(* Logix 5000 project; controller Modbus_TCP_Client_Example vendor 1 type 14 code 154 rev 32.15; software revision 32.05; part 10 of 10 *)
(* tags used below, declared in another part *)
   Transaction : raC_UDT_ModbusClientTransaction;
   Wrk_Bit : DINT;
   Wrk_Byte : DINT;
(* raC_Tec_NetModbusTCPClient_BuildReqStr, continued *)

ROUTINE Prescan   (* ladder *)
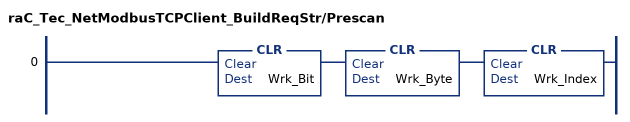
   0: CLR(Wrk_Bit)CLR(Wrk_Byte)CLR(Wrk_Index);
END_ROUTINE
END_ADD_ON_INSTRUCTION

ADD_ON_INSTRUCTION raC_Tec_NetModbusTCPClient_ChkWrReply   (* revision 2.0, ExecutePrescan *)
VAR_OUTPUT
   TransFound : BOOL; {access Read Only}
END_VAR
VAR_IN_OUT
   Transactions : raC_UDT_ModbusClientTransaction[5]; {required}
END_VAR
VAR_INPUT
   TransactionID : INT; {required}
   ModbusBytes : DINT; {required}
END_VAR
VAR_OUTPUT
   LocalOffset : INT; {access Read Only}
   Count : INT; {access Read Only}
END_VAR
VAR_INPUT
   Command : DINT; {required}
   LastTransaction : DINT; {required}
END_VAR
VAR
   Wrk_TransactionPtr : DINT; {access None}
END_VAR

ROUTINE Logic   (* ladder *)
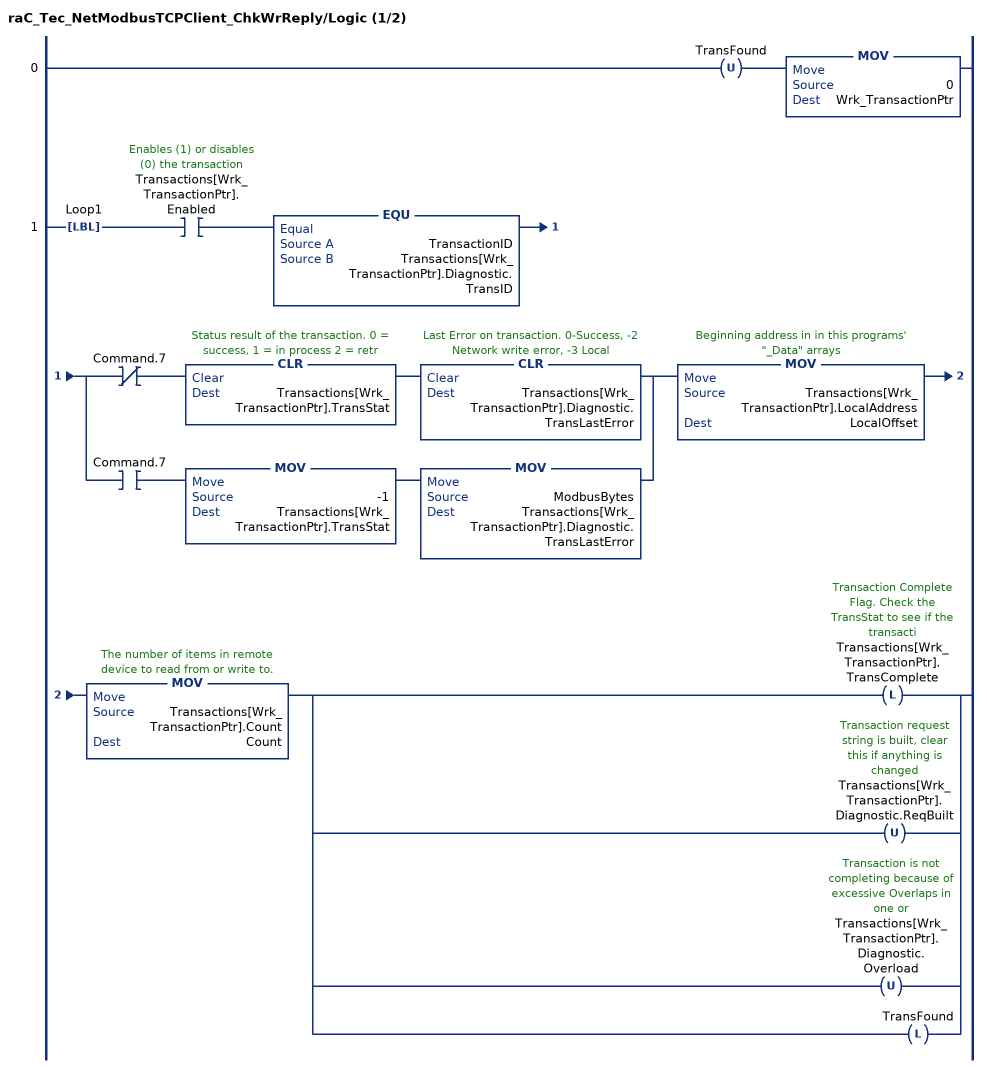
   0: OTU(TransFound)MOV(0,Wrk_TransactionPtr);
   1: LBL(Loop1)XIC(Transactions[Wrk_TransactionPtr].Enabled)EQU(TransactionID,Transactions[Wrk_TransactionPtr].Diagnostic.TransID)[XIO(Command.7) CLR(Transactions[Wrk_TransactionPtr].TransStat) CLR(Transactions[Wrk_TransactionPtr].Diagnostic.TransLastError) ,XIC(Command.7) MOV(-1,Transactions[Wrk_TransactionPtr].TransStat) MOV(ModbusBytes,Transactions[Wrk_TransactionPtr].Diagnostic.TransLastError) ]MOV(Transactions[Wrk_TransactionPtr].LocalAddress,LocalOffset)MOV(Transactions[Wrk_TransactionPtr].Count,Count)[OTL(Transactions[Wrk_TransactionPtr].TransComplete) ,OTU(Transactions[Wrk_TransactionPtr].Diagnostic.ReqBuilt) ,OTU(Transactions[Wrk_TransactionPtr].Diagnostic.Overload) ,OTL(TransFound) ];
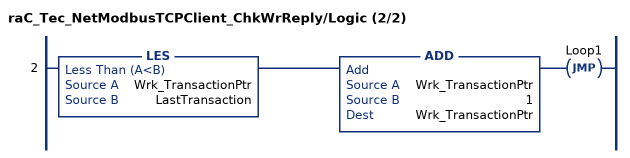
   2: LES(Wrk_TransactionPtr,LastTransaction)ADD(Wrk_TransactionPtr,1,Wrk_TransactionPtr)JMP(Loop1);
END_ROUTINE

ROUTINE Prescan   (* ladder *)
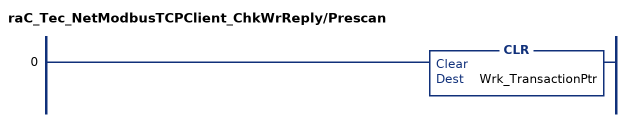
   0: CLR(Wrk_TransactionPtr);
END_ROUTINE
END_ADD_ON_INSTRUCTION

ADD_ON_INSTRUCTION raC_Tec_NetModbusTCPClient_RespStrBit   (* revision 2.0, ExecutePrescan *)
VAR_INPUT
   Inputs : BOOL; {required}
   Modbus_CMD_Len : INT; {required}
   LocalOffset : INT; {required}
END_VAR
VAR_IN_OUT
   ModbusData : raC_UDT_ModbusClientData; {required}
   CommandString : STR0500; {required}
END_VAR
VAR
   Wrk_BufferByteIndex : DINT; {access None}
   Wrk_Cmd_Last : INT; {access None}
   Wrk_Index : DINT; {access None}
   Wrk_BufferBitIndex : DINT; {access None}
   Wrk_ArraySize : DINT; {access None}
END_VAR

ROUTINE Logic   (* ladder *)
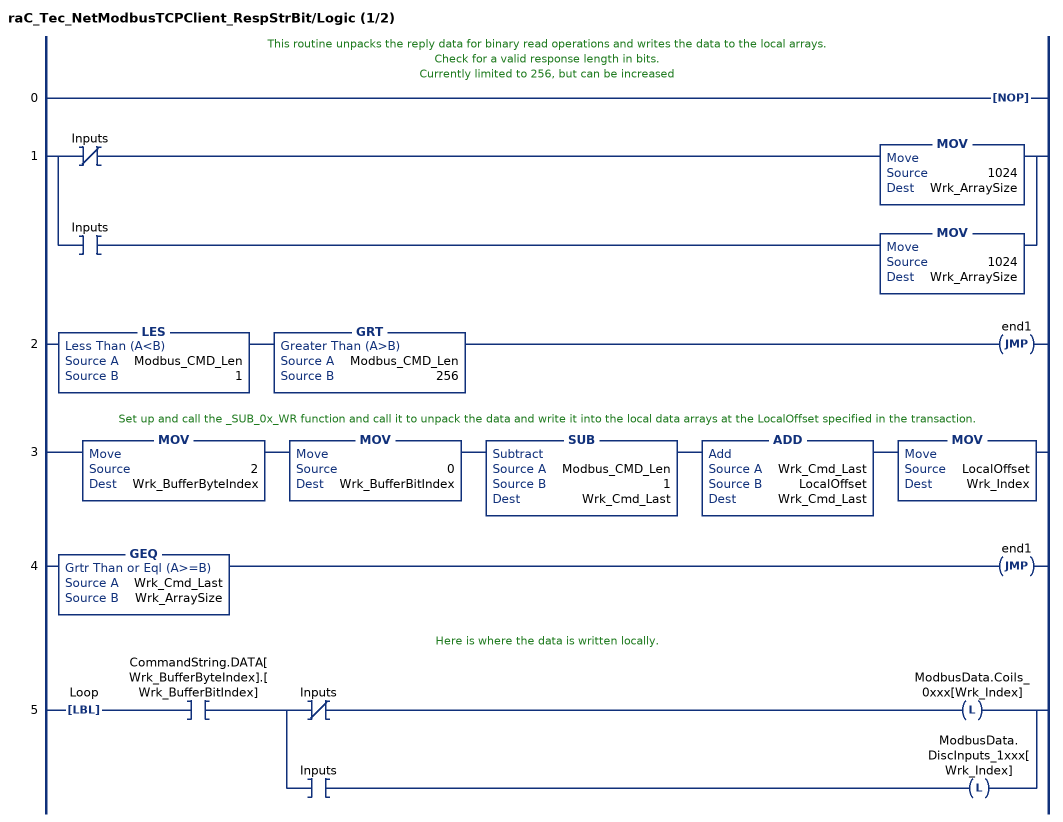
   // This routine unpacks the reply data for binary read operations and writes the data to the local arrays.
   // Check for a valid response length in bits.
   // Currently limited to 256, but can be increased
   0: NOP();
   1: [XIO(Inputs) MOV(1024,Wrk_ArraySize) ,XIC(Inputs) MOV(1024,Wrk_ArraySize) ];
   2: LES(Modbus_CMD_Len,1)GRT(Modbus_CMD_Len,256)JMP(end1);
   // Set up and call the _SUB_0x_WR function and call it to unpack the data and write it into the local data arrays at the LocalOffset specified in the transaction.
   3: MOV(2,Wrk_BufferByteIndex)MOV(0,Wrk_BufferBitIndex)SUB(Modbus_CMD_Len,1,Wrk_Cmd_Last)ADD(Wrk_Cmd_Last,LocalOffset,Wrk_Cmd_Last)MOV(LocalOffset,Wrk_Index);
   4: GEQ(Wrk_Cmd_Last,Wrk_ArraySize)JMP(end1);
   // Here is where the data is written locally.
   5: LBL(Loop)XIC(CommandString.DATA[Wrk_BufferByteIndex].[Wrk_BufferBitIndex])[XIO(Inputs) OTL(ModbusData.Coils_0xxx[Wrk_Index]) ,XIC(Inputs) OTL(ModbusData.DiscInputs_1xxx[Wrk_Index]) ];
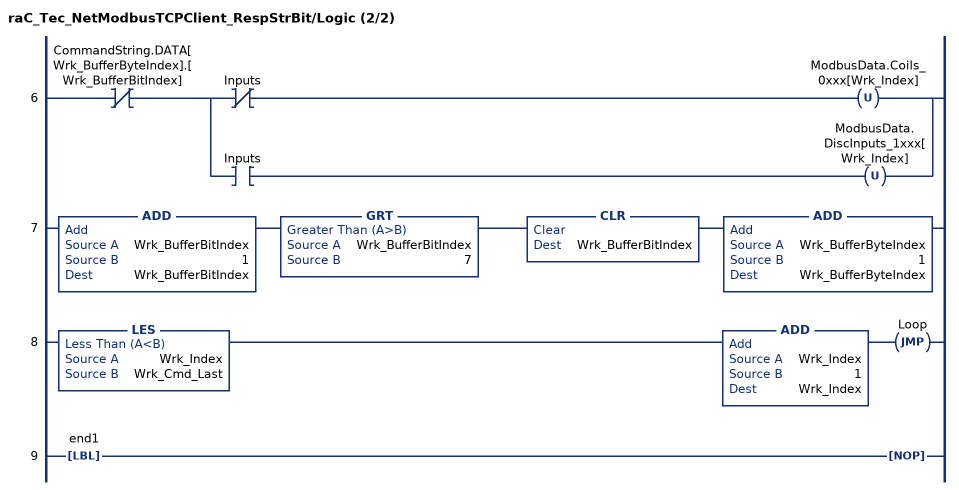
   6: XIO(CommandString.DATA[Wrk_BufferByteIndex].[Wrk_BufferBitIndex])[XIO(Inputs) OTU(ModbusData.Coils_0xxx[Wrk_Index]) ,XIC(Inputs) OTU(ModbusData.DiscInputs_1xxx[Wrk_Index]) ];
   7: ADD(Wrk_BufferBitIndex,1,Wrk_BufferBitIndex)GRT(Wrk_BufferBitIndex,7)CLR(Wrk_BufferBitIndex)ADD(Wrk_BufferByteIndex,1,Wrk_BufferByteIndex);
   8: LES(Wrk_Index,Wrk_Cmd_Last)ADD(Wrk_Index,1,Wrk_Index)JMP(Loop);
   9: LBL(end1)NOP();
END_ROUTINE

ROUTINE Prescan   (* ladder *)
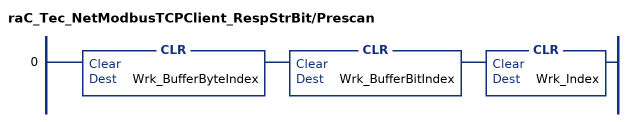
   0: CLR(Wrk_BufferByteIndex)CLR(Wrk_BufferBitIndex)CLR(Wrk_Index);
END_ROUTINE
END_ADD_ON_INSTRUCTION

ADD_ON_INSTRUCTION raC_Tec_NetModbusTCPClient_RespStrWord   (* revision 2.0, ExecutePrescan *)
VAR_INPUT
   Reg3xx : BOOL; {required}
   Modbus_CMD_Len : INT; {required}
   LocalOffset : INT; {required}
END_VAR
VAR_IN_OUT
   ModbusData : raC_UDT_ModbusClientData; {required}
   CommandString : STR0500; {required}
END_VAR
VAR
   Wrk_StringPosition : DINT; {access None}
   Wrk_Cmd_Last : INT; {access None}
   Wrk_Temp_Int : INT; {access None}
   Wrk_Index : DINT; {access None}
END_VAR

ROUTINE Logic   (* ladder *)
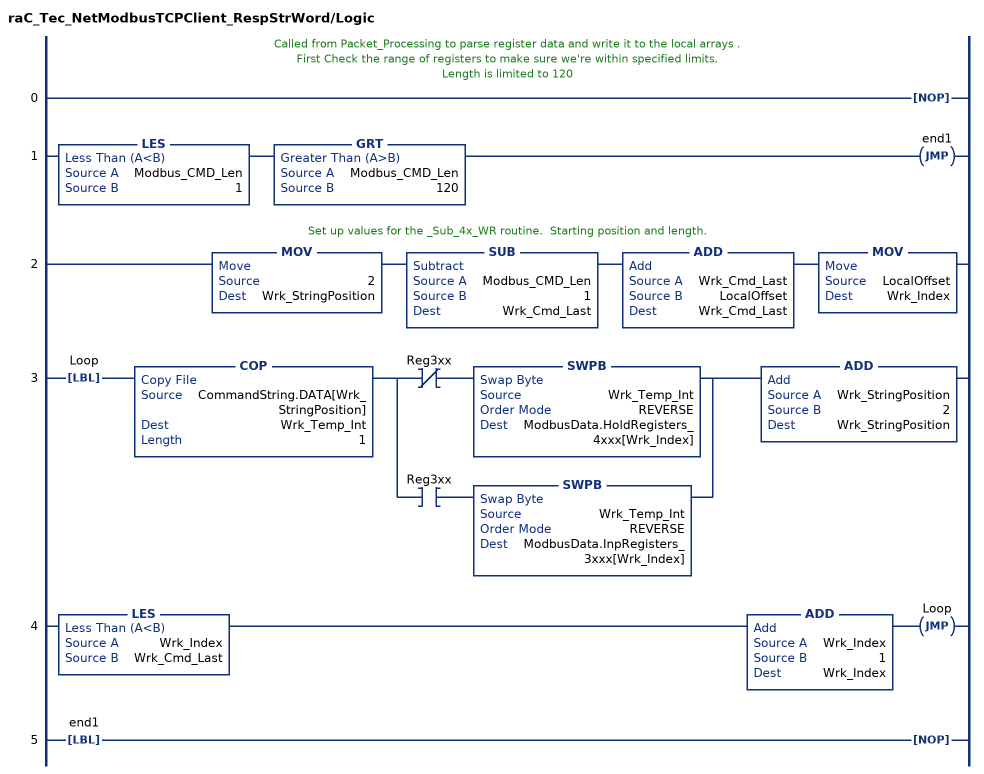
   // Called from Packet_Processing to parse register data and write it to the local arrays .
   // First Check the range of registers to make sure we're within specified limits.
   // Length is limited to 120
   0: NOP();
   1: LES(Modbus_CMD_Len,1)GRT(Modbus_CMD_Len,120)JMP(end1);
   // Set up values for the _Sub_4x_WR routine.  Starting position and length.
   2: MOV(2,Wrk_StringPosition)SUB(Modbus_CMD_Len,1,Wrk_Cmd_Last)ADD(Wrk_Cmd_Last,LocalOffset,Wrk_Cmd_Last)MOV(LocalOffset,Wrk_Index);
   3: LBL(Loop)COP(CommandString.DATA[Wrk_StringPosition],Wrk_Temp_Int,1)[XIO(Reg3xx) SWPB(Wrk_Temp_Int,REVERSE,ModbusData.HoldRegisters_4xxx[Wrk_Index]) ,XIC(Reg3xx) SWPB(Wrk_Temp_Int,REVERSE,ModbusData.InpRegisters_3xxx[Wrk_Index]) ]ADD(Wrk_StringPosition,2,Wrk_StringPosition);
   4: LES(Wrk_Index,Wrk_Cmd_Last)ADD(Wrk_Index,1,Wrk_Index)JMP(Loop);
   5: LBL(end1)NOP();
END_ROUTINE

ROUTINE Prescan   (* ladder *)
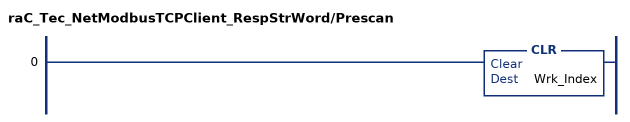
   0: CLR(Wrk_Index);
END_ROUTINE
END_ADD_ON_INSTRUCTION

VAR_GLOBAL   (* controller tags *)
   Alarm_Reset_cmd : BOOL;
   Client_01 : raC_Opr_NetModbusTCPClient := (Inp_Enable := 1, Sts_EN := 1, Sts_Connected := 1, Sts_Overlap := 1);
   Client_01_Data : raC_UDT_ModbusClientData := (HoldRegisters_4xxx[3] := -32751, HoldRegisters_4xxx[4] := 102, HoldRegisters_4xxx[5] := 15, HoldRegisters_4xxx[6] := 753, HoldRegisters_4xxx[7] := -25224, HoldRegisters_4xxx[12] := 338, HoldRegisters_4xxx[13] := 235, HoldRegisters_4xxx[17] := 53, HoldRegisters_4xxx[24] := 82, HoldRegisters_4xxx[27] := 150, HoldRegisters_4xxx[28] := 150, HoldRegisters_4xxx[29] := 2400, HoldRegisters_4xxx[32] := 6, HoldRegisters_4xxx[33] := -32759, HoldRegisters_4xxx[34] := 3, HoldRegisters_4xxx[35] := 15, HoldRegisters_4xxx[36] := 2, HoldRegisters_4xxx[37] := -27218, HoldRegisters_4xxx[40] := 2, HoldRegisters_4xxx[41] := -27218, HoldRegisters_4xxx[42] := 14, HoldRegisters_4xxx[43] := -3067, HoldRegisters_4xxx[48] := 367, HoldRegisters_4xxx[49] := 323, HoldRegisters_4xxx[51] := 479, HoldRegisters_4xxx[55] := 29, HoldRegisters_4xxx[59] := 14, HoldRegisters_4xxx[60] := 1, HoldRegisters_4xxx[61] := 1, HoldRegisters_4xxx[63] := 22600, HoldRegisters_4xxx[67] := 21, HoldRegisters_4xxx[71] := 655, HoldRegisters_4xxx[72] := 9, HoldRegisters_4xxx[73] := 72, HoldRegisters_4xxx[124] := 158, HoldRegisters_4xxx[125] := 158, HoldRegisters_4xxx[126] := 158, HoldRegisters_4xxx[201] := 8, HoldRegisters_4xxx[203] := 255, HoldRegisters_4xxx[204] := -1, HoldRegisters_4xxx[205] := -2328, HoldRegisters_4xxx[206] := -1, HoldRegisters_4xxx[207] := -2328, HoldRegisters_4xxx[208] := -1, HoldRegisters_4xxx[209] := -2328, HoldRegisters_4xxx[212] := 334, HoldRegisters_4xxx[213] := 236, HoldRegisters_4xxx[217] := 53, HoldRegisters_4xxx[503] := -32751, HoldRegisters_4xxx[504] := 3, HoldRegisters_4xxx[505] := 15, HoldRegisters_4xxx[506] := 511, HoldRegisters_4xxx[507] := -5397, HoldRegisters_4xxx[510] := 511, HoldRegisters_4xxx[511] := -5570, HoldRegisters_4xxx[512] := 3, HoldRegisters_4xxx[513] := 23333, HoldRegisters_4xxx[516] := 462, HoldRegisters_4xxx[517] := 477, HoldRegisters_4xxx[518] := 380,
        HoldRegisters_4xxx[519] := 331, HoldRegisters_4xxx[521] := 479, HoldRegisters_4xxx[523] := 172, HoldRegisters_4xxx[525] := 29, HoldRegisters_4xxx[529] := 63);
        .HoldRegisters_4xxx[5]   // Digital Input Status (IS)
        .HoldRegisters_4xxx[10]   // Encoder Position (EP)
        .HoldRegisters_4xxx[11]   // Encoder Position (EP)
        .HoldRegisters_4xxx[21]   // Immediate DC Bus Voltage (Unit =0.1V)
        .HoldRegisters_4xxx[50]   // Holding Register address 40125, Command Opcode
        .HoldRegisters_4xxx[17]   // Immediate Target Velocity (IV1) ( Unit =1/240 rps)
        .HoldRegisters_4xxx[18]   // Immediate Drive Temperature (IT) ( Unit =0.1C)
        .HoldRegisters_4xxx[3]   // Status Word, High word
        .HoldRegisters_4xxx[1]   // Alarm Code, High word
        .HoldRegisters_4xxx[4]   // Digital Output Status (IO)
        .HoldRegisters_4xxx[16]   // Immediate Actual Velocity (IV) ( Unit =1/240 rps)
        .HoldRegisters_4xxx[7]   // Immediate Absolute Position (IP)
        .HoldRegisters_4xxx[0]   // Read Holding Register 40001, Alarm Code, low word
        .HoldRegisters_4xxx[2]   // Status Word, low word
        .HoldRegisters_4xxx[6]   // Immediate Absolute Position (IP)
        .HoldRegisters_4xxx[33].0   // Enabled
        .HoldRegisters_4xxx[33].1   // Samping
        .HoldRegisters_4xxx[33].2   // Fault
        .HoldRegisters_4xxx[33].3   // In Position
        .HoldRegisters_4xxx[33].4   // Moving
        .HoldRegisters_4xxx[33].5   // Jogging
   Client_01_EN : BOOL;
   Client_01_MSG_Connect : MESSAGE;
        MessageParameters(ServiceCode := 16#004c, LocalElement := Client_01_Parameters.MSG_Src[0], ...)
   Client_01_MSG_Create : MESSAGE;
        MessageParameters(ServiceCode := 16#004b, LocalElement := Client_01_Parameters.MSG_Src[0], DestinationTag := Client_01_Parameters.MSG_Dest[0], ...)
   Client_01_MSG_Delete : MESSAGE;
        MessageParameters(ServiceCode := 16#004f, ...)
   Client_01_MSG_Read : MESSAGE;
        MessageParameters(ServiceCode := 16#004d, LocalElement := Client_01_Parameters.MSG_Src[0], DestinationTag := Client_01_Parameters.MSG_Dest[0], ...)
   Client_01_MSG_SetSing : MESSAGE;
        MessageParameters(ServiceCode := 16#0010, LocalElement := Client_01_Parameters.MSG_Src[496], ...)
   Client_01_MSG_Write : MESSAGE;
        MessageParameters(ServiceCode := 16#004e, LocalElement := Client_01_Parameters.MSG_Src[0], DestinationTag := Client_01_Parameters.MSG_Dest[0], ...)
   Client_01_Parameters : raC_UDT_ModbusClientConnection := (DestAddress := '10.10.10.19', DestinationPort := 502, MSG_Src[4] := -28, MSG_Src[5] := 1, MSG_Src[12] := 73, MSG_Src[16] := 106, MSG_Src[17] := -35, MSG_Src[21] := 67, MSG_Src[22] := 1, MSG_Src[23] := 16, MSG_Src[24] := 1, MSG_Src[25] := 79, MSG_Src[27] := 30, MSG_Src[28] := 60, MSG_Src[35] := -128, MSG_Src[36] := 17, MSG_Src[38] := 3, MSG_Src[40] := 15, MSG_Src[41] := 1, MSG_Src[42] := -1, MSG_Src[43] := -22, MSG_Src[44] := -21, MSG_Src[49] := 1, MSG_Src[50] := -1, MSG_Src[51] := -22, MSG_Src[52] := 62, MSG_Src[54] := 3, MSG_Src[55] := 91, MSG_Src[56] := 37, MSG_Src[61] := 1, MSG_Src[62] := -50, MSG_Src[63] := 1, MSG_Src[64] := -35, MSG_Src[65] := 1, MSG_Src[66] := 124, MSG_Src[67] := 1, MSG_Src[68] := 75, MSG_Src[71] := 1, MSG_Src[72] := -33, MSG_Src[76] := -84, MSG_Src[80] := 29, MSG_Src[88] := 63, MSG_Src[90] := 2, MSG_Src[91] := 113, MSG_Src[97] := 4, MSG_Src[98] := -80, MSG_Src[114] := 1, MSG_Src[121] := 2, MSG_Src[122] := 88, MSG_Src[123] := 2, MSG_Src[124] := 88, MSG_Src[125] := 1, MSG_Src[126] := 44, MSG_Src[127] := 9, MSG_Src[128] := 96, MSG_Src[496] := 1, MSG_Dest[8] := 21, MSG_Dest[12] := 106, MSG_Dest[13] := -36, MSG_Dest[17] := 6,
        MSG_Dest[18] := 1, MSG_Dest[19] := 16, MSG_Dest[21] := 120, MSG_Dest[23] := 10, MSG_Dest[24] := 106, MSG_Dest[25] := -35, MSG_Dest[29] := 3, MSG_Dest[30] := 1, MSG_Dest[31] := -112, MSG_Dest[32] := 19, MSG_Dest[34] := 2, MSG_Dest[35] := -107, MSG_Dest[36] := -82, MSG_Dest[42] := 2, MSG_Dest[43] := -107, MSG_Dest[44] := -82, MSG_Dest[46] := 14, MSG_Dest[47] := -12, MSG_Dest[57] := 1, MSG_Dest[58] := 111, MSG_Dest[59] := 1, MSG_Dest[60] := 67, MSG_Dest[63] := 1, MSG_Dest[64] := -32, MSG_Dest[72] := 29, MSG_Dest[80] := 14, MSG_Dest[82] := 5, MSG_Dest[84] := 5, MSG_Dest[87] := 88, MSG_Dest[88] := 72, MSG_Dest[96] := 21, MSG_Dest[103] := 2, MSG_Dest[104] := -113, MSG_Dest[106] := 9, MSG_Dest[108] := 72, MSG_Dest[121] := 102, MSG_Dest[122] := -41, MSG_Dest[126] := 6, MSG_Dest[127] := 1, MSG_Dest[128] := 16, MSG_Dest[130] := 120, MSG_Dest[132] := 10, MSG_Dest[133] := 102, MSG_Dest[134] := -40, MSG_Dest[138] := 3, MSG_Dest[139] := 1, MSG_Dest[140] := -112, MSG_Dest[141] := 19, MSG_Dest[142] := 1, MSG_Dest[143] := -31, MSG_Dest[144] := 44, MSG_Dest[145] := -27, MSG_Dest[150] := 1, MSG_Dest[151] := -31, MSG_Dest[152] := 44, MSG_Dest[153] := -38, MSG_Dest[155] := 12, MSG_Dest[156] := 14, MSG_Dest[157] := 82, MSG_Dest[166] := 1,
        MSG_Dest[167] := 121, MSG_Dest[168] := 1, MSG_Dest[169] := 72, MSG_Dest[172] := 1, MSG_Dest[173] := -33, MSG_Dest[174] := -1, MSG_Dest[175] := -1, MSG_Dest[176] := -1, MSG_Dest[177] := -1, MSG_Dest[181] := 29, MSG_Dest[189] := 52, MSG_Dest[191] := 33, MSG_Dest[193] := 32, MSG_Dest[196] := 88, MSG_Dest[197] := 72, MSG_Dest[205] := 21, MSG_Dest[212] := 2, MSG_Dest[213] := -113, MSG_Dest[215] := 9, MSG_Dest[217] := 72, MSG_Dest[230] := 49, MSG_Dest[231] := 98, MSG_Dest[235] := 6, MSG_Dest[236] := 1, MSG_Dest[237] := 16, MSG_Dest[239] := 120, MSG_Dest[241] := 10);
   Client_01_Transactions : raC_UDT_ModbusClientTransaction[5] := ([0].Enabled := 1, [0].PollInterval := 200, [0].TransType := 3, [0].StationID := 1, [0].Count := 50, [0].TransStat := 1, [0].Diagnostic.Request := 'j$DE$00$00$00$06$01$03$00$00$002', [0].Diagnostic.ReqBuilt := 1, [0].Diagnostic.TransID := 27358, [0].Diagnostic.IntervalTimer.PRE := 160, [0].Diagnostic.IntervalTimer.ACC := 179, [0].Diagnostic.IntervalTimer.EN := 1, [0].Diagnostic.IntervalTimer.DN := 1, [0].Diagnostic.NoReplyCounter.PRE := 10, [0].Diagnostic.PendingTimer.PRE := 3000, [0].Diagnostic.PendingTimer.ACC := 239, [0].Diagnostic.PendingTimer.EN := 1, [0].Diagnostic.PendingTimer.TT := 1, [1].Enabled := 1, [1].PollInterval := 200, [1].TransType := 16, [1].StationID := 1, [1].BeginAddress := 120, [1].Count := 10, [1].LocalAddress := 50, [1].TransComplete := 1, [1].Diagnostic.Request := 'j$DC$00$00$00$1B$01$10$00x$00$0A$14$00$00$00$00$00$00$80$11$00$E2$00$0F$02$F1$9Dx$00$00$00$00', [1].Diagnostic.Overlap := 1, [1].Diagnostic.TransID := 27356, [1].Diagnostic.IntervalTimer.PRE := 160, [1].Diagnostic.IntervalTimer.ACC := 179, [1].Diagnostic.IntervalTimer.EN := 1, [1].Diagnostic.IntervalTimer.DN := 1, [1].Diagnostic.NoReplyCounter.PRE := 10, [1].Diagnostic.PendingTimer.PRE := 3000, [2].PollInterval := 1000, [2].Diagnostic.Request := 'j$DD$00$00$00C$01$10$01O$00$1E<$00$00$00$00$00$00$80$11$00$03$00$0F$01$FF$EA$EB$00$00$00$00$01$FF$EA>$00$03[%$00$00$00$00$01$CE$01$DD$01|$01K$00$00$01$DF$00$00$00$AC$00$00$00$1D$00$00$00$00$00$00$00?', [2].Diagnostic.Overlap := 1, [2].Diagnostic.TransID := 27357, [2].Diagnostic.TransLastError := 2, [2].Diagnostic.IntervalTimer.PRE := 160, [2].Diagnostic.IntervalTimer.ACC := 179, [2].Diagnostic.IntervalTimer.EN := 1, [2].Diagnostic.IntervalTimer.DN := 1, [2].Diagnostic.NoReplyCounter.PRE := 10, [2].Diagnostic.PendingTimer.PRE := 3000, [3].PollInterval := 1000, [3].Diagnostic.IntervalTimer.PRE := 960, [3].Diagnostic.IntervalTimer.ACC := 960, [3].Diagnostic.IntervalTimer.EN := 1, [3].Diagnostic.IntervalTimer.DN := 1, [3].Diagnostic.NoReplyCounter.DN := 1, [4].PollInterval := 1000, [4].Diagnostic.Request := ',$1F$00$00$00$06$00$03$00$01$00$0A', [4].Diagnostic.TransID := 11295, [4].Diagnostic.IntervalTimer.PRE := 960, [4].Diagnostic.IntervalTimer.ACC := 979, [4].Diagnostic.IntervalTimer.EN := 1, [4].Diagnostic.IntervalTimer.DN := 1, [4].Diagnostic.NoReplyCounter.PRE := 10,
        [4].Diagnostic.PendingTimer.PRE := 3000);
        [2].BeginAddress   // Beginning address in remote device to read from or write to. - 40335 start
        [2]   // Not Using
        [1]   // Writing Multiple Holding Registers MDX Address 40120
        [0]   // Reading Holding Register MDX Address 40001
        [3]   // Not Using
        [4]   // Not Using
   DC_Voltage : DINT;   // DC Bus Voltage Reading from Holding Register 40022
   Drive_Temperature_C : DINT;   // Drive Temperature Reading from 40019
   Motor_Disable_cmd : BOOL;
   Motor_Enable_cmd : BOOL;
   Motor_Enabled : BOOL;
   Motor_Faulted : BOOL;
   Motor_Jog_cmd : BOOL;
   Motor_Running : BOOL;
   Motor_Stop_cmd : BOOL;
   Opcode_Val : DINT[10];
   Out_Opcode : DINT;   // Opcode writing to MDX 40125 Register
END_VAR

PROGRAM Modbus_Program   (* main routine MODBUS_CLIENT *)

ROUTINE MODBUS_CLIENT   (* ladder *)
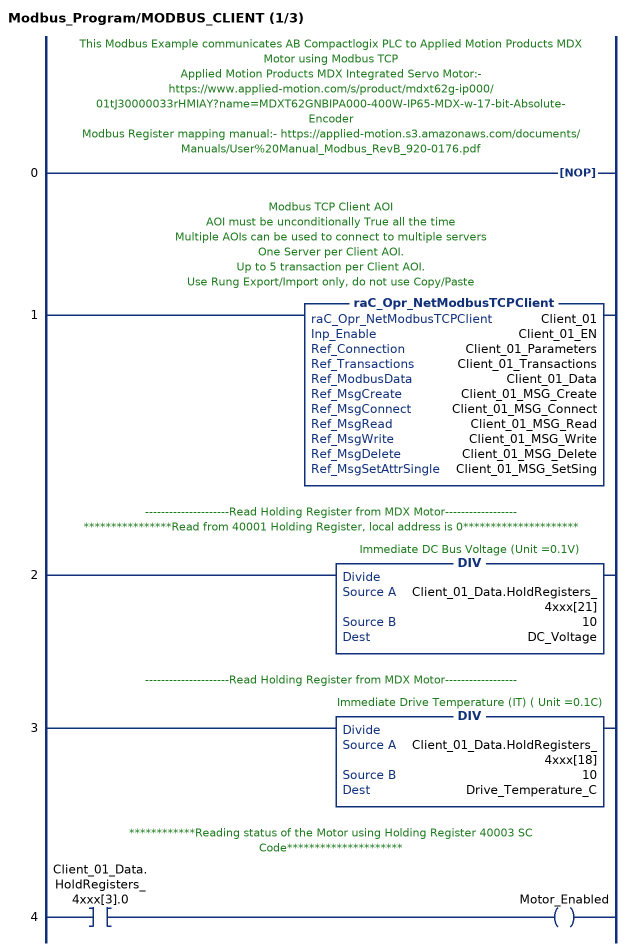
   // This Modbus Example communicates AB Compactlogix PLC to Applied Motion Products MDX Motor using Modbus TCP
   // Applied Motion Products MDX Integrated Servo Motor:- https://www.applied-motion.com/s/product/mdxt62g-ip000/01tJ30000033rHMIAY?name=MDXT62GNBIPA000-400W-IP65-MDX-w-17-bit-Absolute-Encoder
   // Modbus Register mapping manual:- https://applied-motion.s3.amazonaws.com/documents/Manuals/User%20Manual_Modbus_RevB_920-0176.pdf
   0: NOP();
   // Modbus TCP Client AOI
   // AOI must be unconditionally True all the time
   // Multiple AOIs can be used to connect to multiple servers
   // One Server per Client AOI.
   //  Up to 5 transaction per Client AOI.
   // Use Rung Export/Import only, do not use Copy/Paste
   1: raC_Opr_NetModbusTCPClient(Client_01,Client_01_EN,Client_01_Parameters,Client_01_Transactions,Client_01_Data,Client_01_MSG_Create,Client_01_MSG_Connect,Client_01_MSG_Read,Client_01_MSG_Write,Client_01_MSG_Delete,Client_01_MSG_SetSing);
   // ---------------------Read Holding Register from MDX Motor------------------
   // ****************Read from 40001 Holding Register, local address is 0*********************
   2: DIV(Client_01_Data.HoldRegisters_4xxx[21],10,DC_Voltage);
   // ---------------------Read Holding Register from MDX Motor------------------
   3: DIV(Client_01_Data.HoldRegisters_4xxx[18],10,Drive_Temperature_C);
   // ************Reading status of the Motor using Holding Register 40003 SC Code*********************
   4: XIC(Client_01_Data.HoldRegisters_4xxx[3].0)OTE(Motor_Enabled);
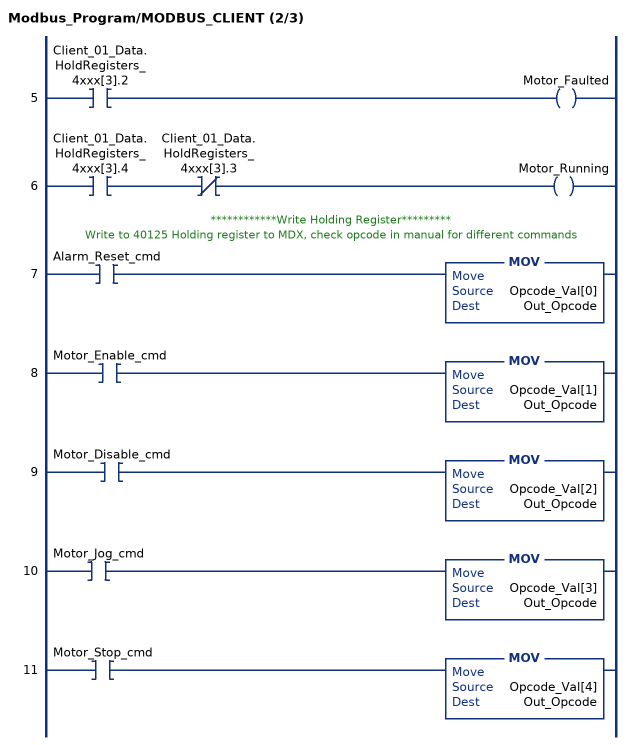
   5: XIC(Client_01_Data.HoldRegisters_4xxx[3].2)OTE(Motor_Faulted);
   6: XIC(Client_01_Data.HoldRegisters_4xxx[3].4)XIO(Client_01_Data.HoldRegisters_4xxx[3].3)OTE(Motor_Running);
   // ************Write Holding Register*********
   // Write to 40125 Holding register to MDX, check opcode in manual for different commands
   7: XIC(Alarm_Reset_cmd)MOV(Opcode_Val[0],Out_Opcode);
   8: XIC(Motor_Enable_cmd)MOV(Opcode_Val[1],Out_Opcode);
   9: XIC(Motor_Disable_cmd)MOV(Opcode_Val[2],Out_Opcode);
   10: XIC(Motor_Jog_cmd)MOV(Opcode_Val[3],Out_Opcode);
   11: XIC(Motor_Stop_cmd)MOV(Opcode_Val[4],Out_Opcode);
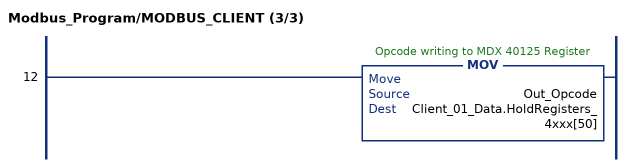
   12: MOV(Out_Opcode,Client_01_Data.HoldRegisters_4xxx[50]);
END_ROUTINE
END_PROGRAM
